{attribute 'GeneratedUsingTerminal: EL3773-0000-0018'}
{attribute addProperty BoxType "EL3773-0000-0018"}
{attribute addProperty Id "EtcSlaveTerminalBaseL1_Voltage_StatusAT %I*L1_Voltage_Status_7371B0437L1_Voltage_SamplesAT %I*L1_Voltage_Samples_926B408D20L1_Current_StatusAT %I*L1_Current_Status_82DECBF67L1_Current_SamplesAT %I*L1_Current_Samples_4D057C4C20L2_Voltage_StatusAT %I*L2_Voltage_Status_0D1813FE7L2_Voltage_SamplesAT %I*L2_Voltage_Samples_A61DC4DD20L2_Current_StatusAT %I*L2_Current_Status_FCB7684B7L2_Current_SamplesAT %I*L2_Current_Samples_7973F81C20L3_Voltage_StatusAT %I*L3_Voltage_Status_273F72957L3_Voltage_SamplesAT %I*L3_Voltage_Samples_B5CFB8ED20L3_Current_StatusAT %I*L3_Current_Status_D69009207L3_Current_SamplesAT %I*L3_Current_Samples_6AA1842C20AI_NextSync1TimeAT %I*AI_NextSync1Time_6DC4D2968AI_Sample_CountAT %I*AI_Sample_Count_EA88CAD92WcStateAT %I*WcState_9091E0EB2InfoDataAT %I*InfoData_BEF6B88E18"}
{attribute addProperty CRC "2975177687"}
{attribute addProperty Size "192"}
TYPE EL3773_B1559BD7 EXTENDS EtcSlaveTerminalBase :
STRUCT
	{attribute addProperty Name "L1_Voltage_Status"}
	L1_Voltage_Status : L1_Voltage_Status_7371B043;
	{attribute addProperty Name "L1_Voltage_Samples"}
	L1_Voltage_Samples : L1_Voltage_Samples_926B408D;
	{attribute addProperty Name "L1_Current_Status"}
	L1_Current_Status : L1_Current_Status_82DECBF6;
	{attribute addProperty Name "L1_Current_Samples"}
	L1_Current_Samples : L1_Current_Samples_4D057C4C;
	{attribute addProperty Name "L2_Voltage_Status"}
	L2_Voltage_Status : L2_Voltage_Status_0D1813FE;
	{attribute addProperty Name "L2_Voltage_Samples"}
	L2_Voltage_Samples : L2_Voltage_Samples_A61DC4DD;
	{attribute addProperty Name "L2_Current_Status"}
	L2_Current_Status : L2_Current_Status_FCB7684B;
	{attribute addProperty Name "L2_Current_Samples"}
	L2_Current_Samples : L2_Current_Samples_7973F81C;
	{attribute addProperty Name "L3_Voltage_Status"}
	L3_Voltage_Status : L3_Voltage_Status_273F7295;
	{attribute addProperty Name "L3_Voltage_Samples"}
	L3_Voltage_Samples : L3_Voltage_Samples_B5CFB8ED;
	{attribute addProperty Name "L3_Current_Status"}
	L3_Current_Status : L3_Current_Status_D6900920;
	{attribute addProperty Name "L3_Current_Samples"}
	L3_Current_Samples : L3_Current_Samples_6AA1842C;
	{attribute addProperty Name "AI_NextSync1Time"}
	AI_NextSync1Time : AI_NextSync1Time_6DC4D296;
	{attribute addProperty Name "AI_Sample_Count"}
	AI_Sample_Count : AI_Sample_Count_EA88CAD9;
	{attribute addProperty Name "WcState"}
	WcState : WcState_9091E0EB;
	{attribute addProperty Name "InfoData"}
	InfoData : InfoData_BEF6B88E;
END_STRUCT
END_TYPE

(* stored: Version 1.2.0.0, ProductVersion 3.1.4024.9
   DUT EL3773_B1559BD7: Id {6753e8c2-5542-48b4-a729-5ad6d4fb84fd} *)
